Fanuc KAREL source: kt00484.KL

-- PROVISIONAL review KL for V1013-1; original PC SHA256 0d7b25fe13edd9d933826ff33368d546cc7547a5f420a4de5813a5289ba117ab
-- Incomplete behavior may be omitted. Consult companion uncertainty JSON. Do not deploy.
PROGRAM KT00484
%NOLOCKGROUP
-- UNRESOLVED_DECL P1 type=000101
-- UNRESOLVED_DECL P2 type=000106
-- UNRESOLVED_DECL OUT type=000101
BEGIN
  -- UNRESOLVED_PC offsets 5-20; opcodes 2E,22,32,35
  -- UNRESOLVED_PC offsets 25-54; opcodes 49,49,7E,60,4A
  -- UNRESOLVED_PC offsets 59-63; opcodes 7F
END KT00484
